(* PLC project test_ethercat, Laurent BESSARD test_ethercat 1.0 *)
(* stored: creationDateTime 2011-10-20T19:01:52, modificationDateTime 2026-03-29T01:56:12 *)

PROGRAM Prog
  VAR
    CLOCK AT %QX0.0.4.28672.1 : BOOL;
    GREENLED AT %QX0.0.4.28688.1 : BOOL := TRUE;
    ControlWord AT %QW0.0.3.24640.0 : UINT;
    StatusWord AT %IW0.0.3.24641.0 : UINT;
    Mode AT %QB0.0.3.24672.0 : SINT;
    ModeDisplay AT %IB0.0.3.24673.0 : SINT;
    ActualPosition AT %ID0.0.3.24676.0 : DINT;
    ActualVelocity AT %ID0.0.3.24684.0 : DINT;
    TargetPosition AT %QD0.0.3.24698.0 : DINT;
    TargetVelocity AT %QD0.0.3.24831.0 : DINT;
    DigitalInputs AT %ID0.0.3.24829.0 : UDINT;
    ActualTorque AT %IW0.0.3.24695.0 : INT;
    TargetTorque AT %QW0.0.3.24689.0 : INT;
  END_VAR

            CLOCK := NOT CLOCK;
          
END_PROGRAM

PROGRAM test_MCL
  VAR
    CLOCK : UDINT;
  END_VAR
  VAR
    Axis AT %IW0.0.3.402 : AXIS_REF;
  END_VAR
  VAR
    switch : MC_Power;
    move1 : MC_MoveAbsolute;
    ActualPosition : DINT;
    Valid : BOOL;
    Pn : LREAL;
    Vn : LREAL;
    MC_MoveVelocity0 : MC_MoveVelocity;
    MC_MoveAbsolute0 : MC_MoveAbsolute;
    readpos : MC_ReadActualPosition;
    readspeed : MC_ReadParameter;
    MC_SetPosition0 : MC_SetPosition;
  END_VAR

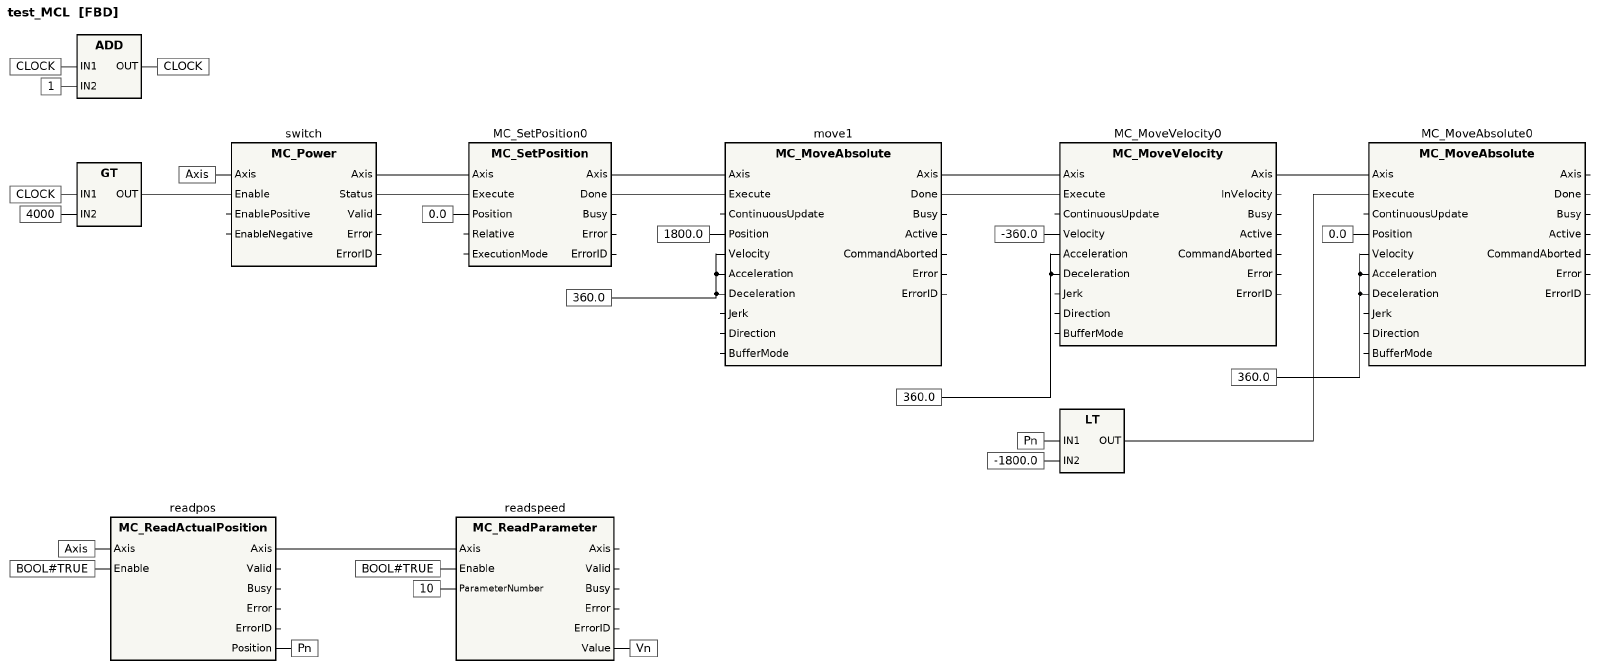
(* FBD diagram, written out as Structured Text *)
CLOCK := CLOCK + 1;
readpos(Axis := Axis, Enable := BOOL#TRUE);
Pn := readpos.Position;
readspeed(Axis := readpos.Axis, Enable := BOOL#TRUE, ParameterNumber := 10);
Vn := readspeed.Value;
switch(Axis := Axis, Enable := CLOCK > 4000);
MC_SetPosition0(Axis := switch.Axis, Execute := switch.Status, Position := 0.0);
move1(Axis := MC_SetPosition0.Axis, Execute := MC_SetPosition0.Done, Position := 1800.0, Velocity := 360.0, Acceleration := 360.0, Deceleration := 360.0);
MC_MoveVelocity0(Axis := move1.Axis, Execute := move1.Done, Velocity := -360.0, Acceleration := 360.0, Deceleration := 360.0);
MC_MoveAbsolute0(Axis := MC_MoveVelocity0.Axis, Execute := Pn < (-1800.0), Position := 0.0, Velocity := 360.0, Acceleration := 360.0, Deceleration := 360.0);
END_PROGRAM

CONFIGURATION conf
  RESOURCE res ON PLC
    TASK main_task(INTERVAL := T#0.5ms, PRIORITY := 0);
    PROGRAM main_instance WITH main_task : Prog;
    PROGRAM test_MCL_instance WITH main_task : test_MCL;
  END_RESOURCE
END_CONFIGURATION
